PROGRAM POU_Contadores
VAR
	iCintaProcesando : INT := 0;
	iStackBoxProcesando: INT := 0;
	iCajaProcesando : INT := 0;
	bGuardandoCaja: BOOL := 0;
	iProcesandoCintas: INT := 0;
	
	reDifSensorSorting: R_TRIG;
	feRRefSensorSortingA: F_TRIG;
	feRRefSensorSortingV: F_TRIG;
	reDifSensorSortingM: F_TRIG;
	fTrigRRefSensorAlmacen: F_TRIG;
	tFTrigEmitterA: F_TRIG;
	tFTrigEmitterV: F_TRIG;
	tFTrigEmitterM: F_TRIG;
	tFTrigDiffuseSensor : F_TRIG;
	
	fFtrigRobotSeMueveA : F_TRIG;
	fFtrigRobotSeMueveV : F_TRIG;
	fFtrigRobotSeMueveM : F_TRIG;
END_VAR

reDifSensorSorting(CLK:= GVL_Sorting.bDiffuseSensorA);
feRRefSensorSortingA(CLK:= GVL_StackBox.bRReflectiveSensorA1);
feRRefSensorSortingV (CLK:= GVL_StackBox.bRReflectiveSensorV1); 
reDifSensorSortingM (CLK:= GVL_Sorting.bDiffuseSensorM);
tFTrigDiffuseSensor(CLK:= GVL_ProcesoPallet.bDiffuseSensorSalida);
fTrigRRefSensorAlmacen(CLK:= GVL_Almacen.bRRflexSensorAlmacen);
tFTrigEmitterA(CLK:= GVL_ProcesoPallet.iLightArrayEmitterA);
tFTrigEmitterV(CLK:= GVL_ProcesoPallet.iLightArrayEmitterV);
tFTrigEmitterM(CLK:= GVL_ProcesoPallet.iLightArrayEmitterM);

fFtrigRobotSeMueveA(CLK:= PRG_PickAndPlace.RobotSeMueveA);
fFtrigRobotSeMueveV(CLK:= PRG_PickAndPlace.RobotSeMueveV);
fFtrigRobotSeMueveM(CLK:= PRG_PickAndPlace.RobotSeMueveM);

// SECCION 1 
(* Sumamos 1 al contador si se comienza a procesar una pieza y se resta 1 cuando se termina de procesar *)

IF reDifSensorSorting.Q THEN
	iCintaProcesando := iCintaProcesando + 1;
END_IF

IF feRRefSensorSortingA.Q THEN
	iCintaProcesando := iCintaProcesando - 1;
END_IF

IF feRRefSensorSortingV.Q THEN
	iCintaProcesando := iCintaProcesando - 1;
END_IF

IF reDifSensorSortingM.Q THEN
	iCintaProcesando := iCintaProcesando - 1;
END_IF


// SECCION 2 
(* Sumamos 1 al contador si se comienza a procesar una pieza y se resta 1 cuando se termina de procesar *)

IF feRRefSensorSortingA.Q THEN
	iStackBoxProcesando := iStackBoxProcesando + 1;
END_IF

IF feRRefSensorSortingV.Q THEN
	iStackBoxProcesando := iStackBoxProcesando + 1;
END_IF

IF reDifSensorSortingM.Q THEN
	iStackBoxProcesando := iStackBoxProcesando + 1;
END_IF


IF fFtrigRobotSeMueveA.Q THEN
	iStackBoxProcesando := iStackBoxProcesando - 1;
END_IF

IF fFtrigRobotSeMueveV.Q THEN
	iStackBoxProcesando := iStackBoxProcesando - 1;
END_IF

IF fFtrigRobotSeMueveM.Q THEN
	iStackBoxProcesando := iStackBoxProcesando - 1;
END_IF

// SECCION 3 
(* Sumamos 1 al contador si se comienza a procesar una pieza y se resta 1 cuando se termina de procesar *)

IF tFTrigEmitterV.Q THEN
	iCajaProcesando := iCajaProcesando + 1;
END_IF

IF tFTrigEmitterA.Q THEN
	iCajaProcesando := iCajaProcesando + 1;
END_IF

IF tFTrigEmitterM.Q THEN
	iCajaProcesando := iCajaProcesando + 1;
END_IF

IF tFTrigDiffuseSensor.Q THEN
	iCajaProcesando := iCajaProcesando - 1;
END_IF


// SECCION 4
(* Sumamos 1 al contador si se comienza a procesar una pieza a través de los roller conveyor y restamos cuando termina de procesar *)

IF tFTrigDiffuseSensor.Q THEN
	iProcesandoCintas := iProcesandoCintas + 1;
END_IF

IF fTrigRRefSensorAlmacen.Q THEN
	iProcesandoCintas := iProcesandoCintas - 1;
END_IF


// SECCION 5 
(* Sumamos 1 al contador si se comienza a procesar una pieza y se resta 1 cuando se termina de procesar *)

IF PRG_Almacen.ALMACEN > 1 THEN
	bGuardandoCaja := TRUE;
END_IF

IF PRG_Almacen.ALMACEN < 2 THEN
	bGuardandoCaja := FALSE;
END_IF

END_PROGRAM

(* stored: Version 1.1.0.1, ProductVersion 3.1.4024.12
   POU POU_Contadores: Id {379e697d-f57d-4e98-8ff8-dde695db2a2f}, SpecialFunc None *)
